Omron CX-Programmer project NewProject (CX-Programmer 9.75)

# PLC project01: CP2E-N N

## Program NewProgram1 (cyclic task 0)

### Section Section1

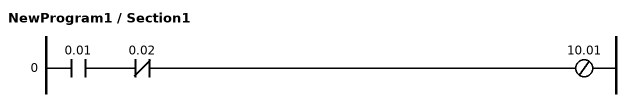
; rung 0
LD 0.01
ANDNOT 0.02
OUTNOT 10.01

### Section END
; rung 0
END(001)